// LS Electric XG5000 project: 최종 plc 프레임_쓰기만 남음
// PLC LSPLC
// module base 0 slot 0: 입출력 모듈:XBC-DR32H (DC 24V 입력, 릴레이 출력 32점)

PROGRAM NewProgram (task: 스캔 프로그램)

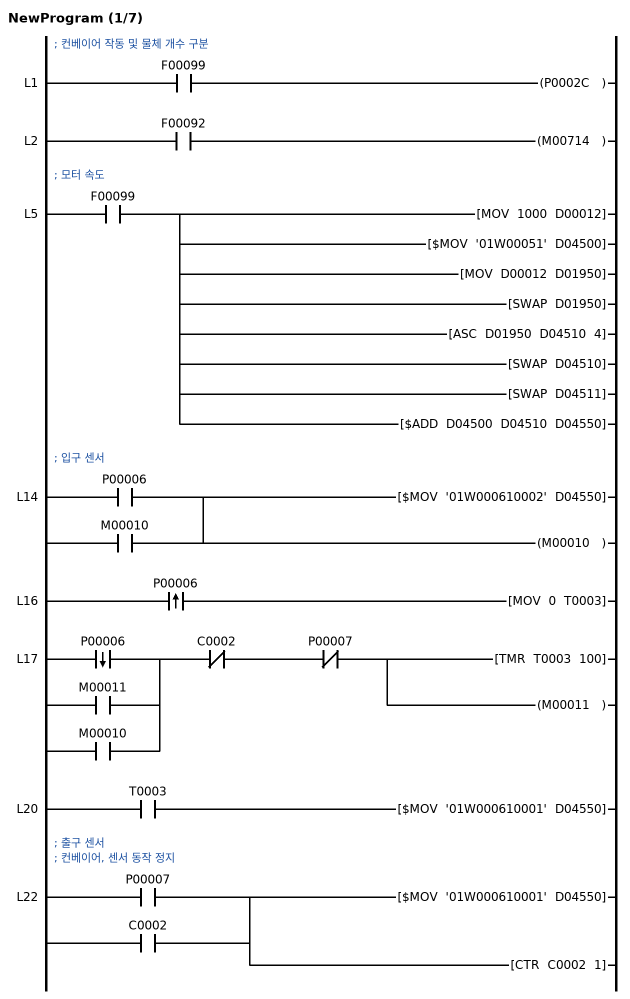
// 컨베이어 작동 및 물체 개수 구분
; L1
LOAD      F00099
OUT       P0002C
; L2
LOAD      F00092
OUT       M00714
// 모터 속도
; L5
LOAD      F00099
MOV       1000 D00012
$MOV      '01W00051' D04500
MOV       D00012 D01950
SWAP      D01950
ASC       D01950 D04510 4
SWAP      D04510
SWAP      D04511
$ADD      D04500 D04510 D04550
// 입구 센서
; L14
LOAD      P00006
OR        M00010
$MOV      '01W000610002' D04550
OUT       M00010
; L16
LOADP     P00006
MOV       0 T0003
; L17
LOADN     P00006
OR        M00011
OR        M00010
AND NOT   C0002
AND NOT   P00007
TMR       T0003 100
OUT       M00011
; L20
LOAD      T0003
$MOV      '01W000610001' D04550
// 출구 센서
; L22
LOAD      P00007
OR        C0002
$MOV      '01W000610001' D04550
CTR       C0002 1
// output comment: 컨베이어, 센서 동작 정지

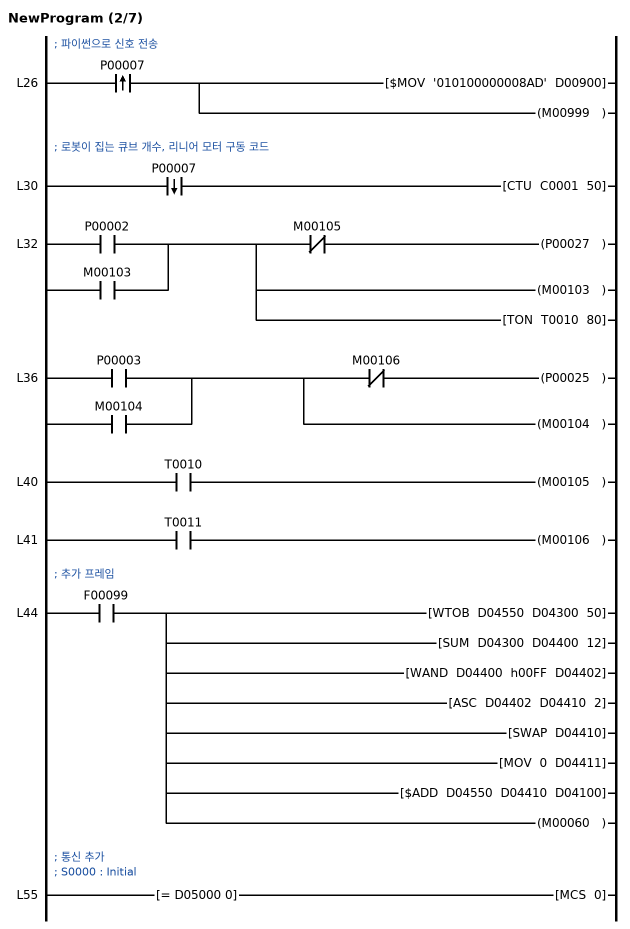
; L26
LOADP     P00007
$MOV      '010100000008AD' D00900
OUT       M00999
// output comment: 파이썬으로 신호 전송
// 로봇이 집는 큐브 개수, 리니어 모터 구동 코드
; L30
LOADN     P00007
CTU       C0001 50
; L32
LOAD      P00002
OR        M00103
MPUSH
AND NOT   M00105
OUT       P00027
MPOP
OUT       M00103
TON       T0010 80
; L36
LOAD      P00003
OR        M00104
MPUSH
AND NOT   M00106
OUT       P00025
MPOP
OUT       M00104
; L40
LOAD      T0010
OUT       M00105
; L41
LOAD      T0011
OUT       M00106
// 추가 프레임
; L44
LOAD      F00099
WTOB      D04550 D04300 50
SUM       D04300 D04400 12
WAND      D04400 h00FF D04402
ASC       D04402 D04410 2
SWAP      D04410
MOV       0 D04411
$ADD      D04550 D04410 D04100
OUT       M00060
// 통신 추가
// S0000 : Initial
; L55
LOAD=     D05000 0
MCS       0

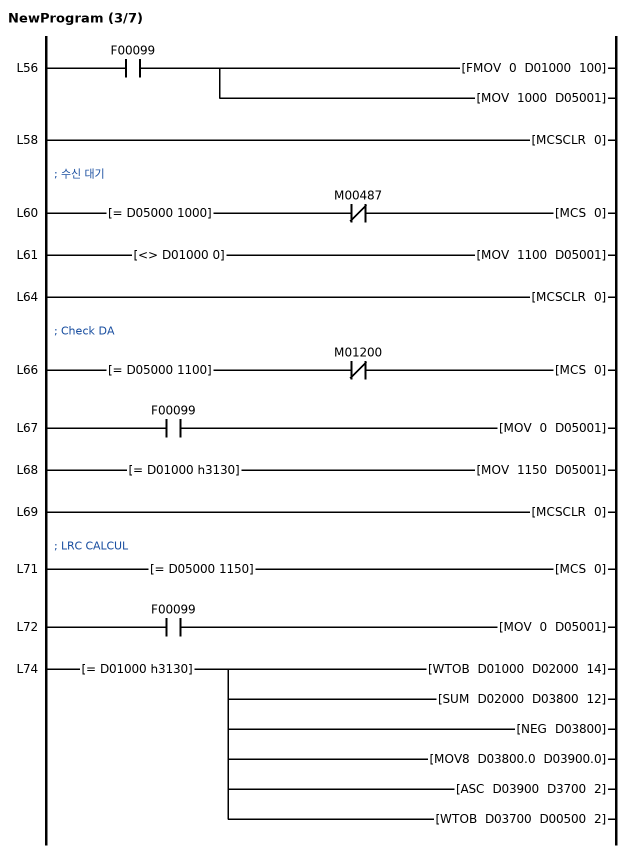
; L56
LOAD      F00099
FMOV      0 D01000 100
MOV       1000 D05001
; L58
MCSCLR    0
// 수신 대기
; L60
LOAD=     D05000 1000
AND NOT   M00487
MCS       0
; L61
LOAD<>    D01000 0
MOV       1100 D05001
; L64
MCSCLR    0
// Check DA
; L66
LOAD=     D05000 1100
AND NOT   M01200
MCS       0
; L67
LOAD      F00099
MOV       0 D05001
; L68
LOAD=     D01000 h3130
MOV       1150 D05001
; L69
MCSCLR    0
// LRC CALCUL
; L71
LOAD=     D05000 1150
MCS       0
; L72
LOAD      F00099
MOV       0 D05001
; L74
LOAD=     D01000 h3130
WTOB      D01000 D02000 14
SUM       D02000 D03800 12
NEG       D03800
MOV8      D03800.0 D03900.0
ASC       D03900 D3700 2
WTOB      D03700 D00500 2

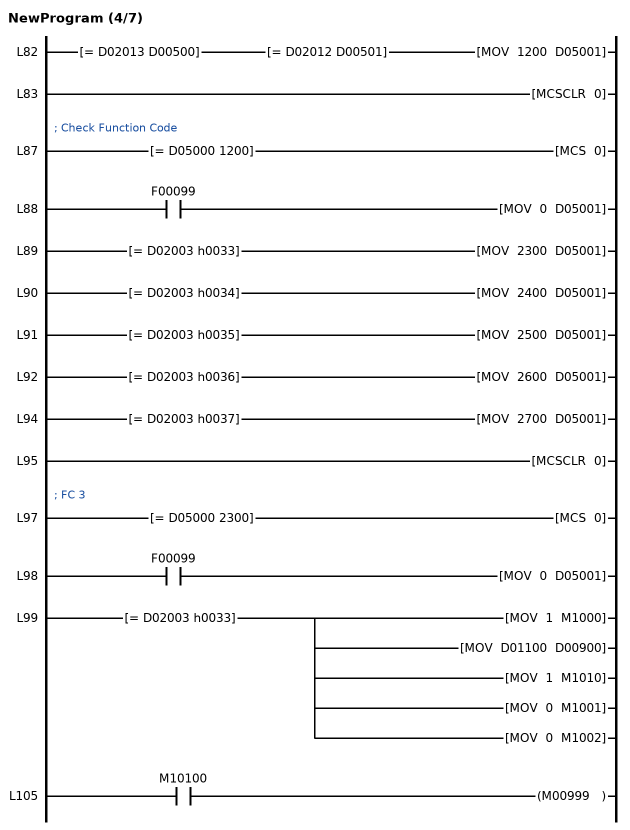
; L82
LOAD=     D02013 D00500
AND=      D02012 D00501
MOV       1200 D05001
; L83
MCSCLR    0
// Check Function Code
; L87
LOAD=     D05000 1200
MCS       0
; L88
LOAD      F00099
MOV       0 D05001
; L89
LOAD=     D02003 h0033
MOV       2300 D05001
; L90
LOAD=     D02003 h0034
MOV       2400 D05001
; L91
LOAD=     D02003 h0035
MOV       2500 D05001
; L92
LOAD=     D02003 h0036
MOV       2600 D05001
; L94
LOAD=     D02003 h0037
MOV       2700 D05001
; L95
MCSCLR    0
// FC 3
; L97
LOAD=     D05000 2300
MCS       0
; L98
LOAD      F00099
MOV       0 D05001
; L99
LOAD=     D02003 h0033
MOV       1 M1000
MOV       D01100 D00900
MOV       1 M1010
MOV       0 M1001
MOV       0 M1002
; L105
LOAD      M10100
OUT       M00999

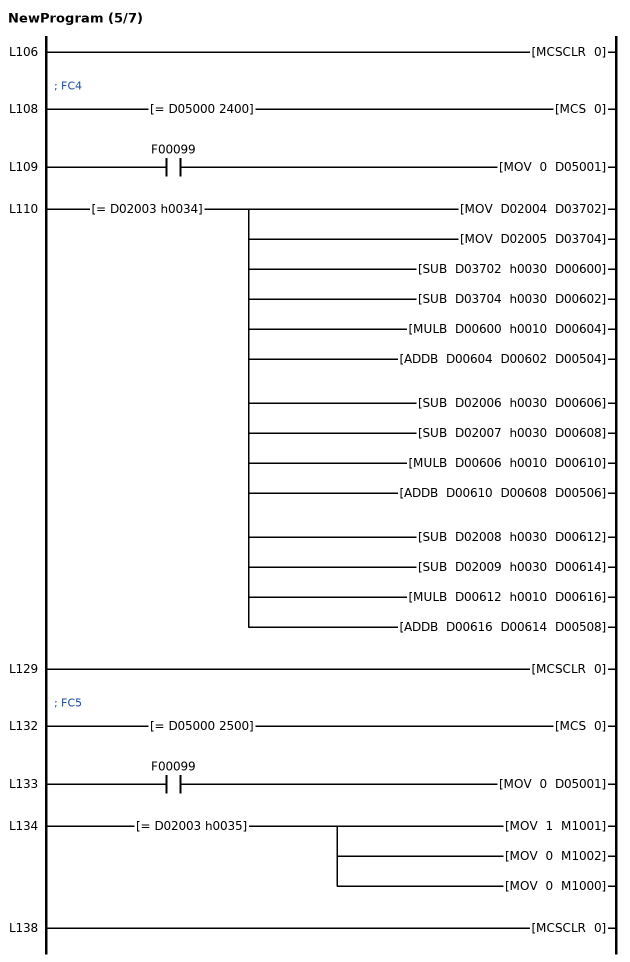
; L106
MCSCLR    0
// FC4
; L108
LOAD=     D05000 2400
MCS       0
; L109
LOAD      F00099
MOV       0 D05001
; L110
LOAD=     D02003 h0034
MOV       D02004 D03702
MOV       D02005 D03704
SUB       D03702 h0030 D00600
SUB       D03704 h0030 D00602
MULB      D00600 h0010 D00604
ADDB      D00604 D00602 D00504
SUB       D02006 h0030 D00606
SUB       D02007 h0030 D00608
MULB      D00606 h0010 D00610
ADDB      D00610 D00608 D00506
SUB       D02008 h0030 D00612
SUB       D02009 h0030 D00614
MULB      D00612 h0010 D00616
ADDB      D00616 D00614 D00508
; L129
MCSCLR    0
// FC5
; L132
LOAD=     D05000 2500
MCS       0
; L133
LOAD      F00099
MOV       0 D05001
; L134
LOAD=     D02003 h0035
MOV       1 M1001
MOV       0 M1002
MOV       0 M1000
; L138
MCSCLR    0

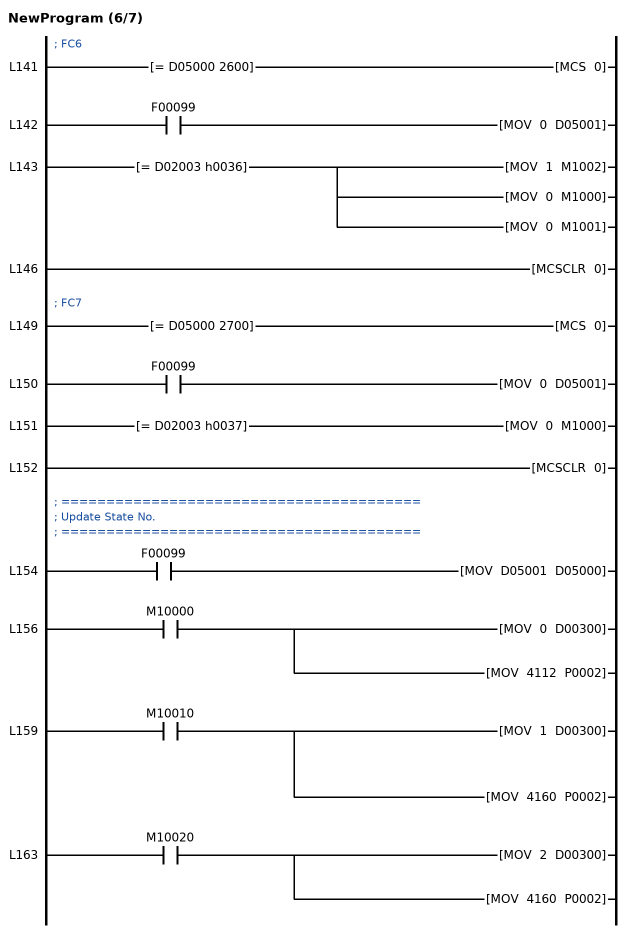
// FC6
; L141
LOAD=     D05000 2600
MCS       0
; L142
LOAD      F00099
MOV       0 D05001
; L143
LOAD=     D02003 h0036
MOV       1 M1002
MOV       0 M1000
MOV       0 M1001
; L146
MCSCLR    0
// FC7
; L149
LOAD=     D05000 2700
MCS       0
; L150
LOAD      F00099
MOV       0 D05001
; L151
LOAD=     D02003 h0037
MOV       0 M1000
; L152
MCSCLR    0
// ========================================
// Update State No.
// ========================================
; L154
LOAD      F00099
MOV       D05001 D05000
; L156
LOAD      M10000
MOV       0 D00300
MOV       4112 P0002
; L159
LOAD      M10010
MOV       1 D00300
MOV       4160 P0002
; L163
LOAD      M10020
MOV       2 D00300
MOV       4160 P0002

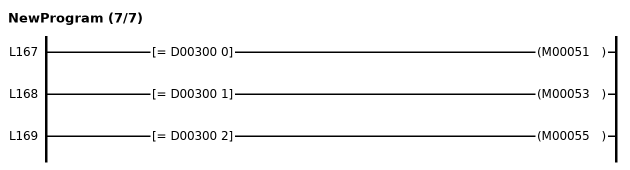
; L167
LOAD=     D00300 0
OUT       M00051
; L168
LOAD=     D00300 1
OUT       M00053
; L169
LOAD=     D00300 2
OUT       M00055